Universal Robots URScript: 180963 (1).script

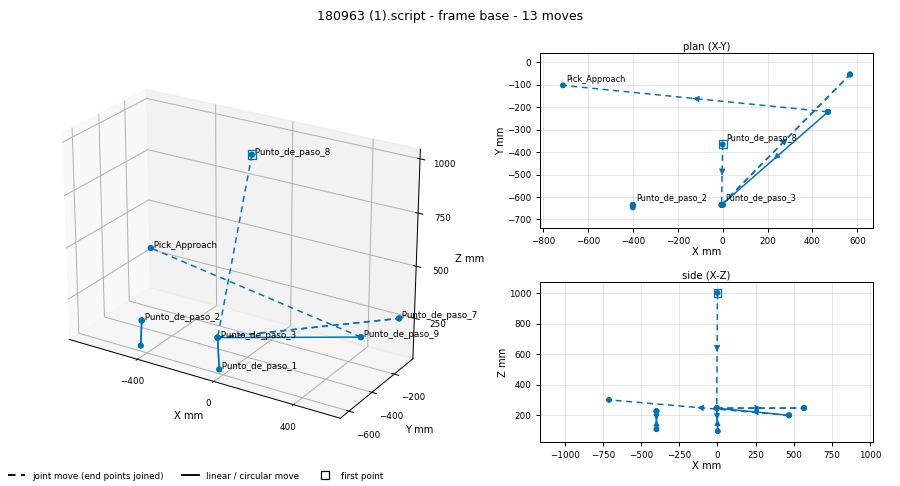
[picture p0: tool path of 180963 (1).script in frame base, 13 of 22 moves have a stored position in this frame; points joined in program order, loops and branches not executed]
def P180963():
  set_tcp(p[0.0,0.0,0.174,0.0,0.0,0.0])
  set_payload(0.92, [0.0, 0.0, 0.058])
  set_tool_voltage(0)
  set_gravity([0.0, 0.0, 9.82])
  set_standard_analog_input_domain(0, 1)
  set_standard_analog_input_domain(1, 1)
  set_tool_analog_input_domain(0, 1)
  set_tool_analog_input_domain(1, 1)
  set_analog_outputdomain(0, 0)
  set_analog_outputdomain(1, 0)
  set_input_actions_to_default()
  step_count_b3da772e_a1e3_478d_8419_95093744ba3c = 0.0
  thread Step_Counter_Thread_0d164cdc_bac2_478b_878c_e3feb41989d4():
    while (True):
      step_count_b3da772e_a1e3_478d_8419_95093744ba3c = step_count_b3da772e_a1e3_478d_8419_95093744ba3c + 1.0
      sync()
    end
  end
  run Step_Counter_Thread_0d164cdc_bac2_478b_878c_e3feb41989d4()
  set_safety_mode_transition_hardness(1)
  global v6=5
  global v5=6
  global v4=5
  global v3=6
  global v2=6
  global v1=5
  global i_var_1__TIMER=0
  global c10=1
  global c9=2
  global c8=2
  global c7=3
  global c6=3
  global c5=3
  global c4=1
  global c3=2
  global c2=2
  global c1=1
  global v10=5
  global v9=7
  global v8=7
  global v7=5
  # begin: URCap Installation Node
  #   Source: External Control, 1.0.5, FZI Research Center for Information Technology
  #   Type: External Control
  # end: URCap Installation Node
  # begin: URCap Installation Node
  #   Source: Robotiq_Grippers, 1.3.1, Robotiq Inc.
  #   Type: Gripper

  ###########################################
  #######Gripper URCap preamble start########
  #######Version null########

  #aliases for the gripper variable names
  ACT = 1
  GTO = 2
  ATR = 3
  ARD = 4
  FOR = 5
  SPE = 6
  OBJ = 7
  STA = 8
  FLT = 9
  POS = 10
  PRE = 11
  LBP = 12
  LRD = 13
  LBL = 14
  LGN = 15

  def rq_init_connection(gripper_sid=9, gripper_socket="1"):
  	socket_open("127.0.0.1",63352, gripper_socket)
  	socket_set_var("SID", gripper_sid,  gripper_socket)
  	ack = socket_read_byte_list(3, gripper_socket)
  end

  def rq_set_sid(gripper_sid=9, gripper_socket="1"):
          socket_set_var("SID", gripper_sid,  gripper_socket)
          sync()
          return is_ack(socket_read_byte_list(3, gripper_socket))
  end

  def rq_activate(gripper_socket="1"):
  	rq_gripper_act = 0

      if (not rq_is_gripper_activated(gripper_socket)):
         rq_reset(gripper_socket)

         while(socket_get_var("ACT",gripper_socket) == 1):
            sleep(0.1)
            rq_reset(gripper_socket)
         end
      end

  	rq_set_var(ACT,1, gripper_socket)
  end

  def rq_activate_and_wait(gripper_socket="1"):
  	rq_activate(gripper_socket)

  	while(not rq_is_gripper_activated(gripper_socket)):
  		# wait for activation completed
  	end
  end

  def rq_stop(gripper_socket="1"):
  	rq_set_var(GTO,0, gripper_socket)
  end

  def rq_reset(gripper_socket="1"):
  	rq_gripper_act = 0
  	rq_obj_detect = 0
  	rq_mov_complete = 0

  	rq_set_var(ACT,0, gripper_socket)
  	rq_set_var(ATR,0, gripper_socket)
  end

  def rq_auto_release_open_and_wait(gripper_socket="1"):
  	rq_set_var(ARD,0, gripper_socket)
  	rq_set_var(ACT,1, gripper_socket)
  	rq_set_var(ATR,1, gripper_socket)

  	gFLT = rq_get_var(FLT, 2, gripper_socket)

  	while(not is_FLT_autorelease_completed(gFLT)):
  		gFLT = rq_get_var(FLT, 2, gripper_socket)
  	end
  end

  def rq_auto_release_close_and_wait(gripper_socket="1"):
  	rq_set_var(ARD,1, gripper_socket)
  	rq_set_var(ACT,1, gripper_socket)
  	rq_set_var(ATR,1, gripper_socket)

  	gFLT = rq_get_var(FLT, 2, gripper_socket)

  	while(not is_FLT_autorelease_completed(gFLT)):
  		gFLT = rq_get_var(FLT, 2, gripper_socket)
  	end
  end

  def rq_set_force(force, gripper_socket="1"):
  	rq_set_var(FOR,force, gripper_socket)
  end

  def rq_set_speed(speed, gripper_socket="1"):
  	rq_set_var(SPE,speed, gripper_socket)
  end

  def rq_open(gripper_socket="1"):
  	rq_move(0, gripper_socket)
  end

  def rq_close(gripper_socket="1"):
  	rq_move(255, gripper_socket)
  end

  def rq_open_and_wait(gripper_socket="1"):
  	rq_move_and_wait(0, gripper_socket)
  end

  def rq_close_and_wait(gripper_socket="1"):
  	rq_move_and_wait(255, gripper_socket)
  end

  def rq_move(pos, gripper_socket="1"):
  	rq_mov_complete = 0
  	rq_obj_detect = 0

  	rq_set_pos(pos, gripper_socket)
  	rq_go_to(gripper_socket)
  end

  def rq_move_and_wait(pos, gripper_socket="1"):
  	rq_move(pos, gripper_socket)

  	while (not rq_is_motion_complete(gripper_socket)):
  		# wait for motion completed
  		sleep(0.01)
  		sync()
  	end

  	# following code used for compatibility with previous versions
  	rq_is_object_detected(gripper_socket)

  	if (rq_obj_detect != 1):
  		rq_mov_complete = 1
  	end
  end

  def rq_wait_for_pos(pos, gripper_socket="1"):
  	gPRE = rq_get_var(PRE, 3, gripper_socket)
  	pre = (gPRE[1] - 48)*100 + (gPRE[2] -48)*10 + gPRE[3] - 48

  	while (pre != pos):
          rq_set_var(POS, pos, gripper_socket)
  		gPRE = rq_get_var(PRE, 3, gripper_socket)
  		pre = (gPRE[1] - 48)*100 + (gPRE[2] -48)*10 + gPRE[3] - 48
  		sync()
  	end

      # Wait for the gripper motion to complete
      while (not rq_is_motion_complete(gripper_socket)):
  		# wait for motion completed
  		sleep(0.01)
  		sync()
  	end

  	# following code used for compatibility with previous versions
  	rq_is_object_detected(gripper_socket)

  	if (rq_obj_detect != 1):
  		rq_mov_complete = 1
  	end
  end

  def rq_wait(gripper_socket="1"):
      # Wait for the gripper motion to complete
      while (not rq_is_motion_complete(gripper_socket)):
  		# wait for motion completed
  		sleep(0.01)
  		sync()
  	end

  	# following code used for compatibility with previous versions
  	rq_is_object_detected(gripper_socket)

  	if (rq_obj_detect != 1):
  		rq_mov_complete = 1
  	end
  end

  def rq_go_to(gripper_socket="1"):
  	rq_set_var(GTO,1, gripper_socket)
  end

  # set the position
  def rq_set_pos(pos, gripper_socket="1"):
  	rq_set_var(POS, pos, gripper_socket)

  	gPRE = rq_get_var(PRE, 3, gripper_socket)
  	pre = (gPRE[1] - 48)*100 + (gPRE[2] -48)*10 + gPRE[3] - 48

  	while (pre != pos):
          rq_set_var(POS, pos, gripper_socket)
  		gPRE = rq_get_var(PRE, 3, gripper_socket)
  		pre = (gPRE[1] - 48)*100 + (gPRE[2] -48)*10 + gPRE[3] - 48
  		sync()
  	end
  end

  # set the position, speed and force
  def rq_set_pos_spd_for(pos, speed, force, gripper_socket="1"):
     rq_send_pos_spd_for(pos, speed, force, gripper_socket)

     ack = socket_read_byte_list(3, gripper_socket)

     while(is_not_ack(ack)):
        rq_send_pos_spd_for(pos, speed, force, gripper_socket)
     	  ack = socket_read_byte_list(3, gripper_socket)
     end
  end

  # send the position, speed and force
  def rq_send_pos_spd_for(pos, speed, force, gripper_socket="1"):

     socket_send_string("SET POS", gripper_socket)
     socket_send_byte(32, gripper_socket)
     socket_send_string(pos, gripper_socket)
     socket_send_byte(32, gripper_socket)
     socket_send_string("SPE", gripper_socket)
     socket_send_byte(32, gripper_socket)
     socket_send_string(speed, gripper_socket)
     socket_send_byte(32, gripper_socket)
     socket_send_string("FOR", gripper_socket)
     socket_send_byte(32, gripper_socket)
     socket_send_string(force, gripper_socket)
     socket_send_byte(10, gripper_socket)

  end

  def rq_is_motion_complete(gripper_socket="1"):
  	rq_mov_complete = 0

  	gOBJ = rq_get_var(OBJ, 1, gripper_socket)
  	sleep(0.01)

  	if (is_OBJ_gripper_at_position(gOBJ)):
  		rq_mov_complete = 1
  		return True
  	end

  	if (is_OBJ_object_detected(gOBJ)):
  		rq_mov_complete = 1
  		return True
  	end

  	return False

  end

  def rq_is_gripper_activated(gripper_socket="1"):
  	gSTA = rq_get_var(STA, 1, gripper_socket)

  	if(is_STA_gripper_activated(gSTA)):
  		rq_gripper_act = 1
  		return True
  	else:
  		rq_gripper_act = 0
  		return False
  	end
  end

  def rq_is_object_detected(gripper_socket="1"):
  	gOBJ = rq_get_var(OBJ, 1, gripper_socket)

  	if(is_OBJ_object_detected(gOBJ)):
  		rq_obj_detect = 1
  		return True
  	else:
  		rq_obj_detect = 0
  		return False
  	end
  end

  def rq_current_pos(gripper_socket="1"):
  	rq_pos = socket_get_var("POS",gripper_socket)
  	sync()
      return rq_pos
  end

  def rq_motor_current(gripper_socket="1"):
  	rq_current = socket_get_var("COU",gripper_socket)
  	sync()
      return rq_current * 10
  end

  def rq_print_gripper_fault_code(gripper_socket="1"):
  	gFLT = rq_get_var(FLT, 2, gripper_socket)

  	if(is_FLT_no_fault(gFLT)):
  		textmsg("Gripper Fault : ", "No Fault (0x00)")
  	elif (is_FLT_action_delayed(gFLT)):
  		textmsg("Gripper Fault : ", "Priority Fault: Action delayed, initialization must be completed prior to action (0x05)")
  	elif (is_FLT_not_activated(gFLT)):
  		textmsg("Gripper Fault : ", "Priority Fault: The activation must be set prior to action (0x07)")
  	elif (is_FLT_autorelease_in_progress(gFLT)):
  		textmsg("Gripper Fault : ", "Minor Fault: Automatic release in progress (0x0B)")
  	elif (is_FLT_overcurrent(gFLT)):
  		textmsg("Gripper Fault : ", "Minor Fault: Overcurrent protection tiggered (0x0E)")
  	elif (is_FLT_autorelease_completed(gFLT)):
  		textmsg("Gripper Fault : ", "Major Fault: Automatic release completed (0x0F)")
  	else:
  		textmsg("Gripper Fault : ", "Unkwown Fault")
  	end
  end

  def rq_print_gripper_num_cycles(gripper_socket="1"):
  	socket_send_string("GET NCY",gripper_socket)
  	sync()
  	string_from_server = socket_read_string(gripper_socket)
  	sync()

  	if(string_from_server == "0"):
  		textmsg("Gripper Cycle Number : ", "Number of cycles is unreachable.")
  	else:
  		textmsg("Gripper Cycle Number : ", string_from_server)
  	end
  end

  def rq_print_gripper_driver_state(gripper_socket="1"):
  	socket_send_string("GET DST",gripper_socket)
  	sync()
  	string_from_server = socket_read_string(gripper_socket)
  	sync()

  	if(string_from_server == "0"):
  		textmsg("Gripper Driver State : ", "RQ_STATE_INIT")
  	elif(string_from_server == "1"):
  		textmsg("Gripper Driver State : ", "RQ_STATE_LISTEN")
  	elif(string_from_server == "2"):
  		textmsg("Gripper Driver State : ", "RQ_STATE_READ_INFO")
  	elif(string_from_server == "3"):
  		textmsg("Gripper Driver State : ", "RQ_STATE_ACTIVATION")
  	else:
  		textmsg("Gripper Driver State : ", "RQ_STATE_RUN")
  	end
  end

  def rq_print_gripper_serial_number(gripper_socket="1"):
  	socket_send_string("GET SNU",gripper_socket)
  	sync()
  	string_from_server = socket_read_string(gripper_socket)
  	sync()
  	textmsg("Gripper Serial Number : ", string_from_server)
  end

  def rq_print_gripper_firmware_version(gripper_socket="1"):
  	socket_send_string("GET FWV",gripper_socket)
  	sync()
  	string_from_server = socket_read_string(gripper_socket)
  	sync()
  	textmsg("Gripper Firmware Version : ", string_from_server)
  end

  def rq_print_gripper_driver_version(gripper_socket="1"):
  	socket_send_string("GET VER",gripper_socket)
  	sync()
  	string_from_server = socket_read_string(gripper_socket)
  	sync()
  	textmsg("Gripper Driver Version : ", string_from_server)
  end

  def rq_print_gripper_probleme_connection(gripper_socket="1"):
  	socket_send_string("GET PCO",gripper_socket)
  	sync()
  	string_from_server = socket_read_string(gripper_socket)
  	sync()
  	if (string_from_server == "0"):
  		textmsg("Gripper Connection State : ", "No connection problem detected")
  	else:
  		textmsg("Gripper Connection State : ", "Connection problem detected")
  	end
  end

  # Returns True if list_of_bytes is [3, 'a', 'c', 'k']
  def is_ack(list_of_bytes):

  	# list length is not 3
  	if (list_of_bytes[0] != 3):
  		return False
  	end

  	# first byte not is 'a'?
  	if (list_of_bytes[1] != 97):
  		return False
  	end

  	# first byte not is 'c'?
  	if (list_of_bytes[2] != 99):
  		return False
  	end

  	# first byte not is 'k'?
  	if (list_of_bytes[3] != 107):
  		return False
  	end

  	return True
  end

  # Returns True if list_of_bytes is not [3, 'a', 'c', 'k']
  def is_not_ack(list_of_bytes):
  	if (is_ack(list_of_bytes)):
  		return False
  	else:
  		return True
  	end
  end

  def is_STA_gripper_activated (list_of_bytes):

  	# list length is not 1
  	if (list_of_bytes[0] != 1):
  		return False
  	end

  	# byte is '3'?
  	if (list_of_bytes[1] == 51):
  		return True
  	end

  	return False
  end

  # Returns True if list_of_byte is [1, '1'] or [1, '2']
  # Used to test OBJ = 0x1 or OBJ = 0x2
  def is_OBJ_object_detected (list_of_bytes):

  	# list length is not 1
  	if (list_of_bytes[0] != 1):
  		return False
  	end

  	# byte is '2'?
  	if (list_of_bytes[1] == 50):
  		return True
  	end

  	# byte is '1'?
  	if (list_of_bytes[1]  == 49):
  		return True
  	end

  	return False

  end

  # Returns True if list_of_byte is [1, '3']
  # Used to test OBJ = 0x3
  def is_OBJ_gripper_at_position (list_of_bytes):

  	# list length is not 1
  	if (list_of_bytes[0] != 1):
  		return False
  	end

  	# byte is '3'?
  	if (list_of_bytes[1] == 51):
  		return True
  	end

  	return False
  end

  def is_not_OBJ_gripper_at_position (list_of_bytes):

  	if (is_OBJ_gripper_at_position(list_of_bytes)):
  		return False
  	else:
  		return True
  	end
  end

  def is_FLT_no_fault(list_of_bytes):

  	# list length is not 2
  	if (list_of_bytes[0] != 2):
  		return False
  	end

  	# first byte is '0'?
  	if (list_of_bytes[1] != 48):
  		return False
  	end

  	# second byte is '0'?
  	if (list_of_bytes[2] != 48):
  		return False
  	end

  	return True

  end

  def is_FLT_action_delayed(list_of_bytes):

  	# list length is not 2
  	if (list_of_bytes[0] != 2):
  		return False
  	end

  	# first byte is '0'?
  	if (list_of_bytes[1] != 48):
  		return False
  	end

  	# second byte is '5'?
  	if (list_of_bytes[2] != 53):
  		return False
  	end

  	return True
  end

  def is_FLT_not_activated(list_of_bytes):

  	# list length is not 2
  	if (list_of_bytes[0] != 2):
  		return False
  	end

  	# first byte is '0'?
  	if (list_of_bytes[1] != 48):
  		return False
  	end

  	# second byte is '7'?
  	if (list_of_bytes[2] != 55):
  		return False
  	end

  	return True
  end

  def is_FLT_autorelease_in_progress(list_of_bytes):

  	# list length is not 2
  	if (list_of_bytes[0] != 2):
  		return False
  	end

  	# first byte is '1'?
  	if (list_of_bytes[1] != 49):
  		return False
  	end

  	# second byte is '1'?
  	if (list_of_bytes[2] != 49):
  		return False
  	end

  	return True

  end

  def is_FLT_overcurrent(list_of_bytes):

  	# list length is not 2
  	if (list_of_bytes[0] != 2):
  		return False
  	end

  	# first byte is '1'?
  	if (list_of_bytes[1] != 49):
  		return False
  	end

  	# second byte is '4'?
  	if (list_of_bytes[2] != 52):
  		return False
  	end

  	return True

  end

  def is_FLT_autorelease_completed(list_of_bytes):

  	# list length is not 2
  	if (list_of_bytes[0] != 2):
  		return False
  	end

  	# first byte is '1'?
  	if (list_of_bytes[1] != 49):
  		return False
  	end

  	# second byte is '5'?
  	if (list_of_bytes[2] != 53):
  		return False
  	end

  	return True

  end

  def rq_set_var(var_name, var_value, gripper_socket="1"):

  	sync()
  	if (var_name == ACT):
  		socket_set_var("ACT", var_value, gripper_socket)
  	elif (var_name == GTO):
  		socket_set_var("GTO", var_value, gripper_socket)
  	elif (var_name == ATR):
  		socket_set_var("ATR", var_value, gripper_socket)
  	elif (var_name == ARD):
  		socket_set_var("ARD", var_value, gripper_socket)
  	elif (var_name == FOR):
  		socket_set_var("FOR", var_value, gripper_socket)
  	elif (var_name == SPE):
  		socket_set_var("SPE", var_value, gripper_socket)
  	elif (var_name == POS):
  		socket_set_var("POS", var_value, gripper_socket)
  	elif (var_name == LBP):
  		socket_set_var("LBP", var_value, gripper_socket)
  	elif (var_name == LRD):
  		socket_set_var("LRD", var_value, gripper_socket)
  	elif (var_name == LBL):
  		socket_set_var("LBL", var_value, gripper_socket)
  	elif (var_name == LGN):
  		socket_set_var("LGN", var_value, gripper_socket)
  	else:
  	end

      sync()

  	ack = socket_read_byte_list(3, gripper_socket)

  	sync()

  	while(is_not_ack(ack)):
  		textmsg("Retry in rq_set_var")

  		textmsg("rq_set_var : retry", " ...")
  		textmsg("rq_set_var : var_name = ", var_name)
  		textmsg("rq_set_var : var_value = ", var_value)

  		if (ack[0] != 0):
  			textmsg("rq_set_var : invalid ack value = ", ack)
  		end

  		socket_set_var(var_name , var_value,gripper_socket)
  		sync()
  		ack = socket_read_byte_list(3, gripper_socket)
  		sync()
  	end
  end


  def rq_get_var(var_name, nbr_bytes, gripper_socket="1"):

  	if (var_name == FLT):
  		socket_send_string("GET FLT",gripper_socket)
  		sync()
  	elif (var_name == OBJ):
  		socket_send_string("GET OBJ",gripper_socket)
  		sync()
  	elif (var_name == STA):
  		socket_send_string("GET STA",gripper_socket)
  		sync()
  	elif (var_name == PRE):
  		socket_send_string("GET PRE",gripper_socket)
  		sync()
  	else:
  	end

  	var_value = socket_read_byte_list(nbr_bytes, gripper_socket)
  	sync()

  	return var_value
  end

  def rq_is_object_validated(gripper_selected, gripper_socket="1"):
  	if(gripper_selected):
  		if(rq_is_object_detected(gripper_socket)):
  		    return True
  		else:
  		    return False
  		end
  	else:
  		return True
  	end
  end

  ############################################
  # normalized functions (maps 0-100 to 0-255)
  ############################################
  def rq_set_force_norm(force_norm, gripper_socket="1"):
      force_gripper = norm_to_gripper(force_norm)
      rq_set_force(force_gripper, gripper_socket)
  end

  def rq_set_speed_norm(speed_norm, gripper_socket="1"):
      speed_gripper = norm_to_gripper(speed_norm)
      rq_set_speed(speed_gripper, gripper_socket)
  end

  def rq_move_norm(pos_norm, gripper_socket="1"):
      pos_gripper = norm_to_gripper(pos_norm)
      rq_move(pos_gripper, gripper_socket)
  end

  def rq_move_and_wait_norm(pos_norm, gripper_socket="1"):
      pos_gripper = norm_to_gripper(pos_norm)
      rq_move_and_wait(pos_gripper, gripper_socket)
  end

  def rq_set_pos_norm(pos_norm, gripper_socket="1"):
      pos_gripper = norm_to_gripper(pos_norm)
      rq_set_pos(pos_gripper, gripper_socket)
  end


  def rq_current_pos_norm(gripper_socket="1"):
      pos_gripper = rq_current_pos(gripper_socket)
      pos_norm = gripper_to_norm(pos_gripper)
      return pos_norm
  end

  def gripper_to_norm(value_gripper):
      value_norm = (value_gripper / 255) * 100
      return floor(value_norm)
  end

  def norm_to_gripper(value_norm):
      value_gripper = (value_norm / 100) * 255
      return ceil(value_gripper)
  end

  def rq_get_position():
      return rq_current_pos_norm()
  end

  def rq_gripper_led_on(gripper_socket="1"):
      rq_set_var(LBP,0, gripper_socket)
  end

  def rq_gripper_led_off(gripper_socket="1"):
      rq_set_var(LBP,1, gripper_socket)
      rq_set_var(LRD,0, gripper_socket)
      rq_set_var(LBL,0, gripper_socket)
      rq_set_var(LGN,0, gripper_socket)
  end

  def rq_gripper_led_force_red(gripper_socket="1"):
      rq_set_var(LBP,1, gripper_socket)
      rq_set_var(LRD,1, gripper_socket)
      rq_set_var(LBL,0, gripper_socket)
      rq_set_var(LGN,0, gripper_socket)
  end

  def rq_gripper_led_force_blue(gripper_socket="1"):
      rq_set_var(LBP,1, gripper_socket)
      rq_set_var(LRD,0, gripper_socket)
      rq_set_var(LBL,1, gripper_socket)
      rq_set_var(LGN,0, gripper_socket)
  end

  def rq_gripper_led_force_green(gripper_socket="1"):
      rq_set_var(LBP,1, gripper_socket)
      rq_set_var(LRD,0, gripper_socket)
      rq_set_var(LBL,0, gripper_socket)
      rq_set_var(LGN,1, gripper_socket)
  end

  def rq_gripper_led_force_purple(gripper_socket="1"):
      rq_set_var(LBP,1, gripper_socket)
      rq_set_var(LRD,1, gripper_socket)
      rq_set_var(LBL,1, gripper_socket)
      rq_set_var(LGN,0, gripper_socket)
  end

  ############################################
  # mm/inches functions
  ############################################
  gripper_closed_norm = [100, 100, 100, 100]
  gripper_open_norm = [0, 0, 0, 0]
  gripper_closed_mm = [0, 0, 0, 0]
  gripper_open_mm = [50, 50, 50, 50]

  def rq_current_pos_mm(gripper_socket=1):
      pos_gripper = rq_current_pos(gripper_socket)
      pos_mm = gripper_to_mm(pos_gripper, gripper_socket)
      return round_value_2_dec(pos_mm)
  end

  def rq_current_pos_inches(gripper_socket=1):
      pos_gripper = rq_current_pos(gripper_socket)
      pos_mm = gripper_to_mm(pos_gripper, gripper_socket)
      pos_in = pos_mm / 25.4
      return round_value_2_dec(pos_in)
  end

  def get_closed_norm(gripper_socket):
      return gripper_closed_norm[gripper_socket - 1]
  end

  def get_open_norm(gripper_socket):
      return gripper_open_norm[gripper_socket - 1]
  end

  def get_closed_mm(gripper_socket):
      return gripper_closed_mm[gripper_socket - 1]
  end

  def get_open_mm(gripper_socket):
      return gripper_open_mm[gripper_socket - 1]
  end

  def set_closed_norm(closed_norm, gripper_socket):
      gripper_closed_norm[gripper_socket - 1] = closed_norm
  end

  def set_open_norm(open_norm, gripper_socket):
      gripper_open_norm[gripper_socket - 1] = open_norm
  end

  def set_closed_mm(closed_mm, gripper_socket):
      gripper_closed_mm[gripper_socket - 1] = closed_mm
  end

  def set_open_mm(open_mm, gripper_socket):
      gripper_open_mm[gripper_socket - 1] = open_mm
  end

  def gripper_to_mm(value_gripper, gripper_socket):
      closed_norm = get_closed_norm(gripper_socket)
      open_norm = get_open_norm(gripper_socket)
      closed_mm = get_closed_mm(gripper_socket)
      open_mm = get_open_mm(gripper_socket)

      value_norm = (value_gripper / 255) * 100

      slope = (closed_mm - open_mm) / (closed_norm - open_norm)
      value_mm = slope * (value_norm - closed_norm) + closed_mm

      if (value_mm > open_mm):
      	value_mm_limited = open_mm
      elif (value_mm < closed_mm):
      	value_mm_limited = closed_mm
      else:
          value_mm_limited = value_mm
      end

      return value_mm_limited
  end

  def round_value(value):
      value_mod = value % 1

  	if(value_mod < 0.5):
  		return floor(value)
  	else:
  		return ceil(value)
  	end
  end

  def round_value_2_dec(value):
      value_x_100 = value * 100
      value_x_100_rounded = round_value(value_x_100)
      return value_x_100_rounded / 100
  end
  #########################################


  rq_obj_detect = 0
  rq_init_connection(9, "1")
  connectivity_checked = [-1,-1,-1,-1]
  status_checked = [-1,-1,-1,-1]
  current_speed = [-1,-1,-1,-1]
  current_force = [-1,-1,-1,-1]
  set_closed_norm(90.19607843137256,1)
  set_open_norm(1.1764705882352942, 1)
  set_closed_mm(0.0, 1)
  set_open_mm(85.0, 1)
  set_closed_norm(100.0,2)
  set_open_norm(0.0, 2)
  set_closed_mm(0.0, 2)
  set_open_mm(50.0, 2)
  set_closed_norm(100.0,3)
  set_open_norm(0.0, 3)
  set_closed_mm(0.0, 3)
  set_open_mm(50.0, 3)
  set_closed_norm(100.0,4)
  set_open_norm(0.0, 4)
  set_closed_mm(0.0, 4)
  set_open_mm(50.0, 4)

  #######Gripper URCap preamble end##########
  ###########################################

  # end: URCap Installation Node
  global cont_1=0
  global cont_2=0
  global cont_3=0
  thread EventThread():
    while (True):
      if (get_standard_digital_in(0) ==   True  ):
        $ 95 "Esperar: 1.0"
        sleep(1.0)
        $ 96 "Ajustar DO[4]=Apagar"
        set_standard_digital_out(4, False)
      elif (get_standard_digital_in(0) ==   False  ):
        $ 98 "Ajustar DO[4]=Encender"
        set_standard_digital_out(4, True)
      end
      sync()
    end
  end
  eventThread = run EventThread()
  while (True):
    $ 1 "Programa de robot"
    $ 2 "Ajustar DO[4]=Encender"
    set_standard_digital_out(4, True)
    $ 3 "Ajustar"
    set_payload(0.92)
    $ 4 "MoverJ"
    $ 5 "Punto_de_paso_8" "breakAfter"
    movej(get_inverse_kin(p[-.000019524487, -.365449998802, 1.001059001102, .000066671487, 2.221363147326, -2.221363159013], qnear=[-3.5587941304981996E-5, -1.570796314870016, 4.8160552978515625E-5, -1.5707481543170374, 8.388957940042019E-5, 1.1984225238848012E-5]), a=1.3962634015954636, v=1.0471975511965976)
    $ 6 "Bucle 48 veces"
    Bucle_1 = 0
    while (Bucle_1 < 48):
      $ 7 "Esperar: 0.5"
      sleep(0.5)
      $ 8 "If digital_in[0]≟ True "
      if (get_standard_digital_in(0) ==   True  ):
        # begin: URCap Program Node
        #   Source: Robotiq_Grippers, 1.3.1, Robotiq Inc.
        #   Type: Gripper
        $ 9 "Gripper Open (1)"
        gripper_1_used = True
        if (connectivity_checked[0] != 1):
          if not(rq_set_sid(9, "1")):
            popup("Gripper 1 must be connected to run this program.", "No connection", False, True, True)
          end
          connectivity_checked[0] = 1
        end
        if (status_checked[0] != 1):
          if not(rq_is_gripper_activated("1")):
            popup("Gripper 1 is not activated. Go to Installation tab > Gripper to activate it and run the program again.", "Not activated", False, True, True)
          end
          status_checked[0] = 1
        end
        rq_set_speed(255, "1")
        current_speed[0] = 255
        rq_set_force(255, "1")
        current_force[0] = 255
        rq_set_pos(0, "1")
        rq_go_to("1")
        rq_wait("1")
        gripper_1_selected = True
        gripper_2_selected = False
        gripper_3_selected = False
        gripper_4_selected = False
        gripper_1_used = False
        gripper_2_used = False
        gripper_3_used = False
        gripper_4_used = False
        # end: URCap Program Node
        $ 10 "MoverJ"
        $ 11 "Punto_de_paso_3" "breakAfter"
        movej(get_inverse_kin(p[-.004983795435, -.634850671169, .245361417840, 2.218933385213, 2.188364492207, .016317964645], qnear=[1.3792614936828613, -1.2451031843768519, 1.2215752601623535, -1.5527899901019495, -1.544217888508932, 1.3932065963745117]), a=1.3962634015954636, v=1.0471975511965976)
        $ 12 "MoverL"
        $ 13 "Punto_de_paso_1" "breakAfter"
        movel(p[.002281377344, -.634850583716, .093823248840, 2.218880177050, 2.188400560307, .016336928912], a=1.2, v=0.25)
        # begin: URCap Program Node
        #   Source: Robotiq_Grippers, 1.3.1, Robotiq Inc.
        #   Type: Gripper
        $ 14 "Gripper Close (1)"
        gripper_1_used = True
        if (connectivity_checked[0] != 1):
          if not(rq_set_sid(9, "1")):
            popup("Gripper 1 must be connected to run this program.", "No connection", False, True, True)
          end
          connectivity_checked[0] = 1
        end
        if (status_checked[0] != 1):
          if not(rq_is_gripper_activated("1")):
            popup("Gripper 1 is not activated. Go to Installation tab > Gripper to activate it and run the program again.", "Not activated", False, True, True)
          end
          status_checked[0] = 1
        end
        rq_set_speed(0, "1")
        current_speed[0] = 0
        rq_set_force(153, "1")
        current_force[0] = 153
        rq_set_pos(255, "1")
        rq_go_to("1")
        rq_wait("1")
        gripper_1_selected = True
        gripper_2_selected = False
        gripper_3_selected = False
        gripper_4_selected = False
        gripper_1_used = False
        gripper_2_used = False
        gripper_3_used = False
        gripper_4_used = False
        # end: URCap Program Node
        $ 15 "If digital_in[1]≟ True "
        if (get_standard_digital_in(1) ==   True  ):
          $ 16 "MoverL"
          $ 17 "Punto_de_paso_6" "breakAfter"
          movel(p[-.004985401254, -.634861247665, .245397363864, 2.218905727147, 2.188235842238, .016231811947], a=1.2, v=0.25)
          $ 18 "MoverJ"
          $ 19 "Punto_de_paso_7" "breakAfter"
          movej(get_inverse_kin(p[.567495628410, -.053997257006, .245389759575, -.006263447627, 3.131128411057, .039609140831], qnear=[2.8415980339050293, -1.4036710898028772, 1.4211440086364746, -1.5904911200152796, -1.5436065832721155, 1.2668311595916748]), a=1.3962634015954636, v=1.0471975511965976)
          $ 20 "Palé"
          cont_2_x_ratio = (cont_2%3)/2
          cont_2_y_ratio = (floor(cont_2/3)%2)/1
          cont_2_z_ratio = (floor(cont_2/6))/1
          pose_2 = interpolate_pose(interpolate_pose(interpolate_pose(p[.567492969880, .154672328125, .005869977308, -.006151930623, 3.131135114152, .039650778495], p[.567480864694, -.125891846128, .005806900340, -.006352381333, 3.131274375057, .039591625587], cont_2_x_ratio), interpolate_pose(p[.641872892390, .156688994744, .005890260992, -.006231708049, 3.131114325923, .039620248473], p[.641890203837, -.125922605385, .005884267350, -.006234417715, 3.131047186433, .039608225966], cont_2_x_ratio), cont_2_y_ratio), interpolate_pose(interpolate_pose(p[.567526646379, .154636886575, .045047983976, -.006433893392, 3.131007760578, .039472178898], p[.567493074625, -.125893200148, .045003067318, -.006429051227, 3.131203550852, .039520061848], cont_2_x_ratio), interpolate_pose(p[.641821170634, .156669009873, .044995270636, -.006304533949, 3.131207511437, .039461988946], p[.641799949895, -.125864206128, .045060158560, -.006303130184, 3.131326550755, .039826230196], cont_2_x_ratio), cont_2_y_ratio), cont_2_z_ratio)
          if (cont_2 >= 11):
            cont_2 = 0
          else:
            cont_2 = cont_2 + 1
          end
          $ 31 "Acercar_3" "noBreak"
          movel(pose_trans(pose_2, pose_trans(pose_inv(p[.567434816893, .154690560631, .005816975098, -.006129744092, 3.131301743890, .039561227546]),p[.567452978940, .154684917029, .064661232932, -.006132505776, 3.131152345937, .039574723348])), a=1.2, v=0.25)
          $ 32 "PuntoDePatrón_3" "noBreak"
          movel(pose_2, a=1.2, v=0.25)
          # begin: URCap Program Node
          #   Source: Robotiq_Grippers, 1.3.1, Robotiq Inc.
          #   Type: Gripper
          $ 33 "Gripper Move42mm (1)" "noBreak"
          gripper_1_used = True
          if (connectivity_checked[0] != 1):
            if not(rq_set_sid(9, "1")):
              popup("Gripper 1 must be connected to run this program.", "No connection", False, True, True)
            end
            connectivity_checked[0] = 1
          end
          if (status_checked[0] != 1):
            if not(rq_is_gripper_activated("1")):
              popup("Gripper 1 is not activated. Go to Installation tab > Gripper to activate it and run the program again.", "Not activated", False, True, True)
            end
            status_checked[0] = 1
          end
          rq_set_speed(0, "1")
          current_speed[0] = 0
          rq_set_force(0, "1")
          current_force[0] = 0
          rq_set_pos(118, "1")
          rq_go_to("1")
          rq_wait("1")
          gripper_1_selected = True
          gripper_2_selected = False
          gripper_3_selected = False
          gripper_4_selected = False
          gripper_1_used = False
          gripper_2_used = False
          gripper_3_used = False
          gripper_4_used = False
          # end: URCap Program Node
          $ 34 "Ajustar" "noBreak"
          set_payload(0.92)
          $ 35 "Esperar: 0.5" "noBreak"
          sleep(0.5)
          $ 36 "Salir_3" "noBreak"
          movel(pose_trans(pose_2, pose_trans(pose_inv(p[.567434816893, .154690560631, .005816975098, -.006129744092, 3.131301743890, .039561227546]),p[.567480217868, .154661499922, .152312951734, -.006096492882, 3.131085752503, .039636744415])), a=1.2, v=0.25)
          $ 37 "MoverJ"
          $ 38 "Punto_de_paso_9" "breakAfter"
          movej(get_inverse_kin(p[.469428746337, -.220494067585, .198063982018, -.006014554298, 3.131287459041, .039491365638], qnear=[2.4772486686706543, -1.5119765440570276, 1.6614856719970703, -1.712616268788473, -1.5447567144977015, 0.9025106430053711]), a=1.3962634015954636, v=1.0471975511965976)
        else:
          $ 39 "Else" "noBreak"
          $ 40 "MoverL"
          $ 41 "Punto_de_paso_6" "breakAfter"
          movel(p[-.004985401254, -.634861247665, .245397363864, 2.218905727147, 2.188235842238, .016231811947], a=1.2, v=0.25)
          $ 42 "MoverJ"
          $ 43 "Punto_de_paso_7" "breakAfter"
          movej(get_inverse_kin(p[.567495628410, -.053997257006, .245389759575, -.006263447627, 3.131128411057, .039609140831], qnear=[2.8415980339050293, -1.4036710898028772, 1.4211440086364746, -1.5904911200152796, -1.5436065832721155, 1.2668311595916748]), a=1.3962634015954636, v=1.0471975511965976)
          $ 44 "Palé"
          cont_3_x_ratio = (cont_3%3)/2
          cont_3_y_ratio = (floor(cont_3/3)%2)/1
          cont_3_z_ratio = (floor(cont_3/6))/1
          pose_3 = interpolate_pose(interpolate_pose(interpolate_pose(p[.757453782070, .154617557121, .005731016151, -.006096576893, 3.131338355623, .039588255529], p[.757491663814, -.125876806229, .005857519520, -.005688303077, 3.130975712113, .039552329111], cont_3_x_ratio), interpolate_pose(p[.831939180111, .156528902805, .005989460839, -.006357874559, 3.130933086022, .039402533660], p[.831743096648, -.125808411147, .005829509205, -.007160338788, 3.131526542281, .039944163084], cont_3_x_ratio), cont_3_y_ratio), interpolate_pose(interpolate_pose(p[.757615953570, .154448324184, .045088945191, -.005821976001, 3.130888991608, .039427400206], p[.757443027519, -.125774501103, .045169480760, -.005778645967, 3.131145737677, .039702401859], cont_3_x_ratio), interpolate_pose(p[.831888331229, .156461545753, .044950244589, -.006223512298, 3.131169142466, .039481219416], p[.831751046053, -.125821131964, .045007880717, -.005359252584, 3.131584806456, .039972518636], cont_3_x_ratio), cont_3_y_ratio), cont_3_z_ratio)
          if (cont_3 >= 11):
            cont_3 = 0
          else:
            cont_3 = cont_3 + 1
          end
          $ 55 "Acercar_2" "noBreak"
          movel(pose_trans(pose_3, pose_trans(pose_inv(p[.757450738307, .154663163544, .005788766890, -.006043107931, 3.131146772158, .039489747696]),p[.757496438800, .154628836054, .072144129680, -.006175492910, 3.131086591061, .039492030587])), a=1.2, v=0.25)
          $ 56 "PuntoDePatrón_2" "noBreak"
          movel(pose_3, a=1.2, v=0.25)
          # begin: URCap Program Node
          #   Source: Robotiq_Grippers, 1.3.1, Robotiq Inc.
          #   Type: Gripper
          $ 57 "Gripper Move42mm (1)" "noBreak"
          gripper_1_used = True
          if (connectivity_checked[0] != 1):
            if not(rq_set_sid(9, "1")):
              popup("Gripper 1 must be connected to run this program.", "No connection", False, True, True)
            end
            connectivity_checked[0] = 1
          end
          if (status_checked[0] != 1):
            if not(rq_is_gripper_activated("1")):
              popup("Gripper 1 is not activated. Go to Installation tab > Gripper to activate it and run the program again.", "Not activated", False, True, True)
            end
            status_checked[0] = 1
          end
          rq_set_speed(0, "1")
          current_speed[0] = 0
          rq_set_force(0, "1")
          current_force[0] = 0
          rq_set_pos(118, "1")
          rq_go_to("1")
          rq_wait("1")
          gripper_1_selected = True
          gripper_2_selected = False
          gripper_3_selected = False
          gripper_4_selected = False
          gripper_1_used = False
          gripper_2_used = False
          gripper_3_used = False
          gripper_4_used = False
          # end: URCap Program Node
          $ 58 "Ajustar" "noBreak"
          set_payload(0.92)
          $ 59 "Esperar: 0.5" "noBreak"
          sleep(0.5)
          $ 60 "Salir_2" "noBreak"
          movel(pose_trans(pose_3, pose_trans(pose_inv(p[.757450738307, .154663163544, .005788766890, -.006043107931, 3.131146772158, .039489747696]),p[.757430805529, .154588553127, .062858555465, -.006038912122, 3.131336344478, .039363364445])), a=1.2, v=0.25)
          $ 61 "MoverJ"
          $ 62 "Punto_de_paso_9" "breakAfter"
          movej(get_inverse_kin(p[.469428746337, -.220494067585, .198063982018, -.006014554298, 3.131287459041, .039491365638], qnear=[2.4772486686706543, -1.5119765440570276, 1.6614856719970703, -1.712616268788473, -1.5447567144977015, 0.9025106430053711]), a=1.3962634015954636, v=1.0471975511965976)
        end
      else:
        $ 63 "Else" "noBreak"
        $ 64 "MoverJ"
        $ 65 "Pick_Approach" "breakAfter"
        movej(get_inverse_kin(p[-.711456046454, -.102481442365, .299283792542, -2.231275387535, -2.205229863966, .019411623598], qnear=[-0.011439148579732716, -0.9799864927874964, 0.6895599365234375, -1.292197052632467, -1.5650880972491663, 3.35932825691998E-4]), a=1.3962634015954636, v=1.0471975511965976)
        $ 66 "Ajustar DO[0]=Encender"
        set_standard_digital_out(0, True)
        # begin: URCap Program Node
        #   Source: Robotiq_Grippers, 1.3.1, Robotiq Inc.
        #   Type: Gripper
        $ 67 "Gripper Open (1)"
        gripper_1_used = True
        if (connectivity_checked[0] != 1):
          if not(rq_set_sid(9, "1")):
            popup("Gripper 1 must be connected to run this program.", "No connection", False, True, True)
          end
          connectivity_checked[0] = 1
        end
        if (status_checked[0] != 1):
          if not(rq_is_gripper_activated("1")):
            popup("Gripper 1 is not activated. Go to Installation tab > Gripper to activate it and run the program again.", "Not activated", False, True, True)
          end
          status_checked[0] = 1
        end
        rq_set_speed(255, "1")
        current_speed[0] = 255
        rq_set_force(255, "1")
        current_force[0] = 255
        rq_set_pos(0, "1")
        rq_go_to("1")
        rq_wait("1")
        gripper_1_selected = True
        gripper_2_selected = False
        gripper_3_selected = False
        gripper_4_selected = False
        gripper_1_used = False
        gripper_2_used = False
        gripper_3_used = False
        gripper_4_used = False
        # end: URCap Program Node
        $ 68 "Palé"
        cont_1_x_ratio = (cont_1%3)/2
        cont_1_y_ratio = (floor(cont_1/3)%4)/3
        cont_1_z_ratio = (floor(cont_1/12))/1
        pose_1 = interpolate_pose(interpolate_pose(interpolate_pose(p[-.760191556201, .026650317112, .047770001305, 2.219032799382, 2.188187952042, .016574802258], p[-.760298970054, -.255055342136, .047917838079, 2.219156125136, 2.188448200975, .016046654292], cont_1_x_ratio), interpolate_pose(p[-.556161939858, .026622709814, .047892137825, 2.219111383269, 2.188497797569, .016255022477], p[-.556149261034, -.255133118331, .047815947280, 2.218978939109, 2.188551714403, .016287508458], cont_1_x_ratio), cont_1_y_ratio), interpolate_pose(interpolate_pose(p[-.760179604127, .026620404965, .002786680283, 2.218883626874, 2.188303628578, .016600609767], p[-.760257828972, -.254987186222, .002762421060, 2.219182690024, 2.188261507034, .016530918440], cont_1_x_ratio), interpolate_pose(p[-.556121228507, .026632291460, .002772321050, 2.219135964668, 2.188180400532, .016493918893], p[-.556140284400, -.255085198716, .002721845055, 2.219033733003, 2.188393602368, .016399801877], cont_1_x_ratio), cont_1_y_ratio), cont_1_z_ratio)
        if (cont_1 >= 23):
          cont_1 = 0
        else:
          cont_1 = cont_1 + 1
        end
        $ 79 "Acercar_1" "noBreak"
        movel(pose_trans(pose_1, pose_trans(pose_inv(p[-.760140621841, .026757377168, .044175241029, 2.218695566769, 2.188538527762, .016598222081]),p[-.760241089330, .026613411270, .132617671107, 2.219120035384, 2.188302181154, .016423655774])), a=1.2, v=0.25)
        $ 80 "PuntoDePatrón_1" "noBreak"
        movel(pose_1, a=1.2, v=0.25)
        $ 81 "Ajustar" "noBreak"
        set_payload(1.17)
        # begin: URCap Program Node
        #   Source: Robotiq_Grippers, 1.3.1, Robotiq Inc.
        #   Type: Gripper
        $ 82 "Gripper Close (1)" "noBreak"
        gripper_1_used = True
        if (connectivity_checked[0] != 1):
          if not(rq_set_sid(9, "1")):
            popup("Gripper 1 must be connected to run this program.", "No connection", False, True, True)
          end
          connectivity_checked[0] = 1
        end
        if (status_checked[0] != 1):
          if not(rq_is_gripper_activated("1")):
            popup("Gripper 1 is not activated. Go to Installation tab > Gripper to activate it and run the program again.", "Not activated", False, True, True)
          end
          status_checked[0] = 1
        end
        rq_set_speed(51, "1")
        current_speed[0] = 51
        rq_set_force(153, "1")
        current_force[0] = 153
        rq_set_pos(255, "1")
        rq_go_to("1")
        rq_wait("1")
        gripper_1_selected = True
        gripper_2_selected = False
        gripper_3_selected = False
        gripper_4_selected = False
        gripper_1_used = False
        gripper_2_used = False
        gripper_3_used = False
        gripper_4_used = False
        # end: URCap Program Node
        $ 83 "Esperar: 0.5" "noBreak"
        sleep(0.5)
        $ 84 "Salir_1" "noBreak"
        movel(pose_trans(pose_1, pose_trans(pose_inv(p[-.760140621841, .026757377168, .044175241029, 2.218695566769, 2.188538527762, .016598222081]),p[-.760236861670, .026578742461, .132624273667, 2.219096811812, 2.188277538837, .016347744001])), a=1.2, v=0.25)
        $ 85 "MoverJ"
        $ 86 "Punto_de_paso_2" "breakAfter"
        movej(get_inverse_kin(p[-.400403861737, -.634866641720, .225479782059, 2.219209903608, 2.188089415148, .016259436640], qnear=[0.8532858490943909, -0.9088681379901331, 0.7602262496948242, -1.4136231581317347, -1.545044247304098, 0.8672980070114136]), a=1.3962634015954636, v=1.0471975511965976)
        $ 87 "MoverL"
        $ 88 "Punto_de_paso_4" "breakAfter"
        movel(p[-.400216499587, -.646147186911, .107058176068, 2.219133088420, 2.188314533504, .016645739472], a=1.2, v=0.25)
        # begin: URCap Program Node
        #   Source: Robotiq_Grippers, 1.3.1, Robotiq Inc.
        #   Type: Gripper
        $ 89 "Gripper Open (1)"
        gripper_1_used = True
        if (connectivity_checked[0] != 1):
          if not(rq_set_sid(9, "1")):
            popup("Gripper 1 must be connected to run this program.", "No connection", False, True, True)
          end
          connectivity_checked[0] = 1
        end
        if (status_checked[0] != 1):
          if not(rq_is_gripper_activated("1")):
            popup("Gripper 1 is not activated. Go to Installation tab > Gripper to activate it and run the program again.", "Not activated", False, True, True)
          end
          status_checked[0] = 1
        end
        rq_set_speed(0, "1")
        current_speed[0] = 0
        rq_set_force(153, "1")
        current_force[0] = 153
        rq_set_pos(0, "1")
        rq_go_to("1")
        rq_wait("1")
        gripper_1_selected = True
        gripper_2_selected = False
        gripper_3_selected = False
        gripper_4_selected = False
        gripper_1_used = False
        gripper_2_used = False
        gripper_3_used = False
        gripper_4_used = False
        # end: URCap Program Node
        $ 90 "MoverL"
        $ 91 "Punto_de_paso_5" "breakAfter"
        movel(p[-.400441373131, -.634851284399, .225430293172, 2.219263597184, 2.188008564473, .016390617450], a=1.2, v=0.25)
      end
      Bucle_1 = Bucle_1 + 1
    end
    $ 92 "Ajustar DO[4]=Apagar"
    set_standard_digital_out(4, False)
    $ 93 "Aviso: Pallet terminado. Recolectar Pallets en  Packaging Area y cargar mas  cubos."
    popup("Pallet terminado. Recolectar Pallets en  Packaging Area y cargar mas  cubos.", "Advertencia", True, False, blocking=False)
    halt
  end
end
